PROGRAM Axes_Itp
VAR
	Fb_Axes_ItpLoadProg: ItpLoadProg;
	Fb_Axes_ItpStartStop: ItpStartStop;
	Fb_Axes_BuildItpGoup: CfgBuild3DGroup;
    localstr: STRING;
	localconstr: STRING(255);
	Fb_Axes_ItpReset_Group: ItpReset;
	
	Fb_Axes_ItpReConfig_Group: CfgReconfigGroup;
	Fb_Axes_ItpConfirmHSK: ItpConfirmHsk;
	
	M_code_rtrig: R_TRIG;
	bItpGet_MHsk: bool;
	nItp_MhskNumber: INT;
	nstep: INT;
END_VAR

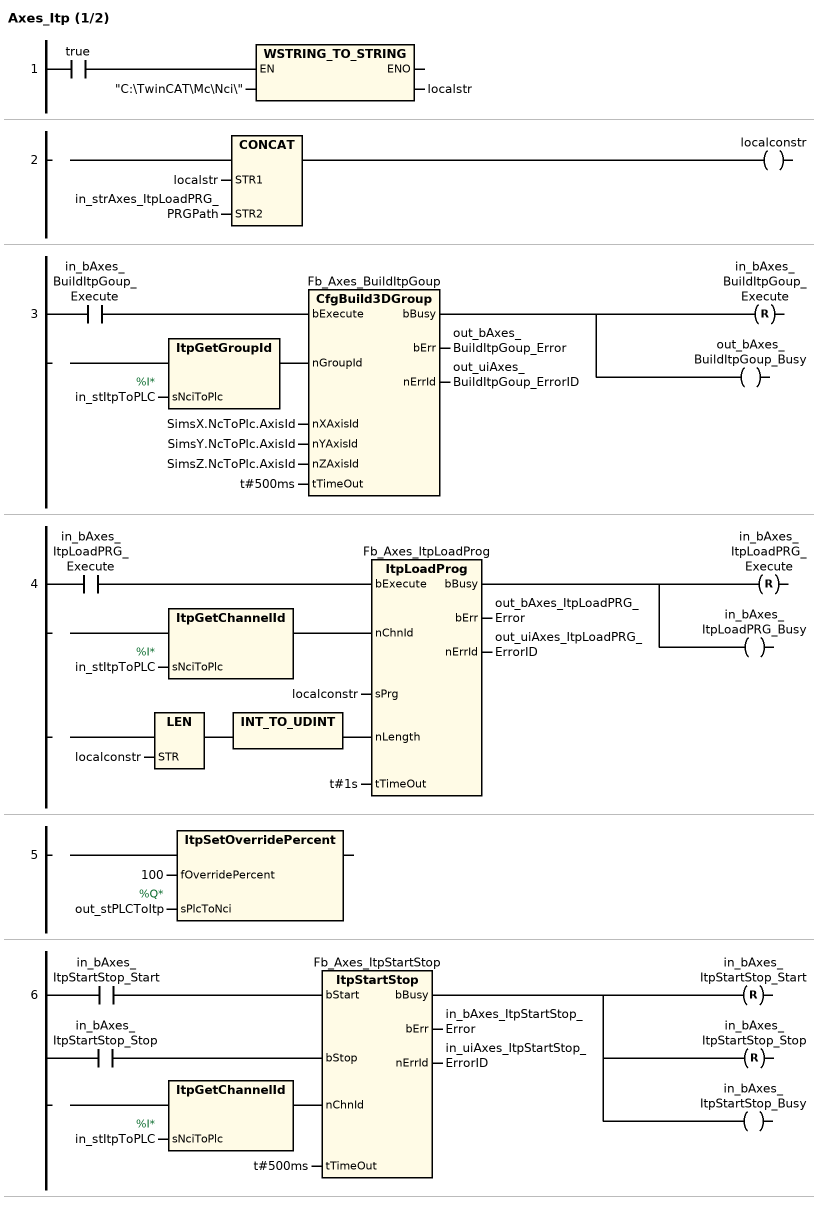
// NETWORK 1
IF true THEN localstr := WSTRING_TO_STRING("C:\TwinCAT\Mc\Nci\"); END_IF

// NETWORK 2
localconstr := CONCAT(STR1 := localstr, STR2 := in_strAxes_ItpLoadPRG_PRGPath);

// NETWORK 3
//   in_stItpToPLC: AT %I*
Fb_Axes_BuildItpGoup(
    bExecute := in_bAxes_BuildItpGoup_Execute,
    nGroupId := ItpGetGroupId(sNciToPlc := in_stItpToPLC),
    nXAxisId := SimsX.NcToPlc.AxisId,
    nYAxisId := SimsY.NcToPlc.AxisId,
    nZAxisId := SimsZ.NcToPlc.AxisId,
    tTimeOut := t#500ms,
    bErr => out_bAxes_BuildItpGoup_Error,
    nErrId => out_uiAxes_BuildItpGoup_ErrorID); // CfgBuild3DGroup
in_bAxes_BuildItpGoup_Execute R= Fb_Axes_BuildItpGoup.bBusy;
out_bAxes_BuildItpGoup_Busy := Fb_Axes_BuildItpGoup.bBusy;

// NETWORK 4
//   in_stItpToPLC: AT %I*
Fb_Axes_ItpLoadProg(
    bExecute := in_bAxes_ItpLoadPRG_Execute,
    nChnId := ItpGetChannelId(sNciToPlc := in_stItpToPLC),
    sPrg := localconstr,
    nLength := INT_TO_UDINT(LEN(STR := localconstr)),
    tTimeOut := t#1s,
    bErr => out_bAxes_ItpLoadPRG_Error,
    nErrId => out_uiAxes_ItpLoadPRG_ErrorID); // ItpLoadProg
in_bAxes_ItpLoadPRG_Execute R= Fb_Axes_ItpLoadProg.bBusy;
in_bAxes_ItpLoadPRG_Busy := Fb_Axes_ItpLoadProg.bBusy;

// NETWORK 5
//   out_stPLCToItp: AT %Q*
ItpSetOverridePercent(fOverridePercent := 100, sPlcToNci := out_stPLCToItp);

// NETWORK 6
//   in_stItpToPLC: AT %I*
Fb_Axes_ItpStartStop(
    bStart := in_bAxes_ItpStartStop_Start,
    bStop := in_bAxes_ItpStartStop_Stop,
    nChnId := ItpGetChannelId(sNciToPlc := in_stItpToPLC),
    tTimeOut := t#500ms,
    bErr => in_bAxes_ItpStartStop_Error,
    nErrId => in_uiAxes_ItpStartStop_ErrorID); // ItpStartStop
in_bAxes_ItpStartStop_Start R= Fb_Axes_ItpStartStop.bBusy;
in_bAxes_ItpStartStop_Stop R= Fb_Axes_ItpStartStop.bBusy;
in_bAxes_ItpStartStop_Busy := Fb_Axes_ItpStartStop.bBusy;

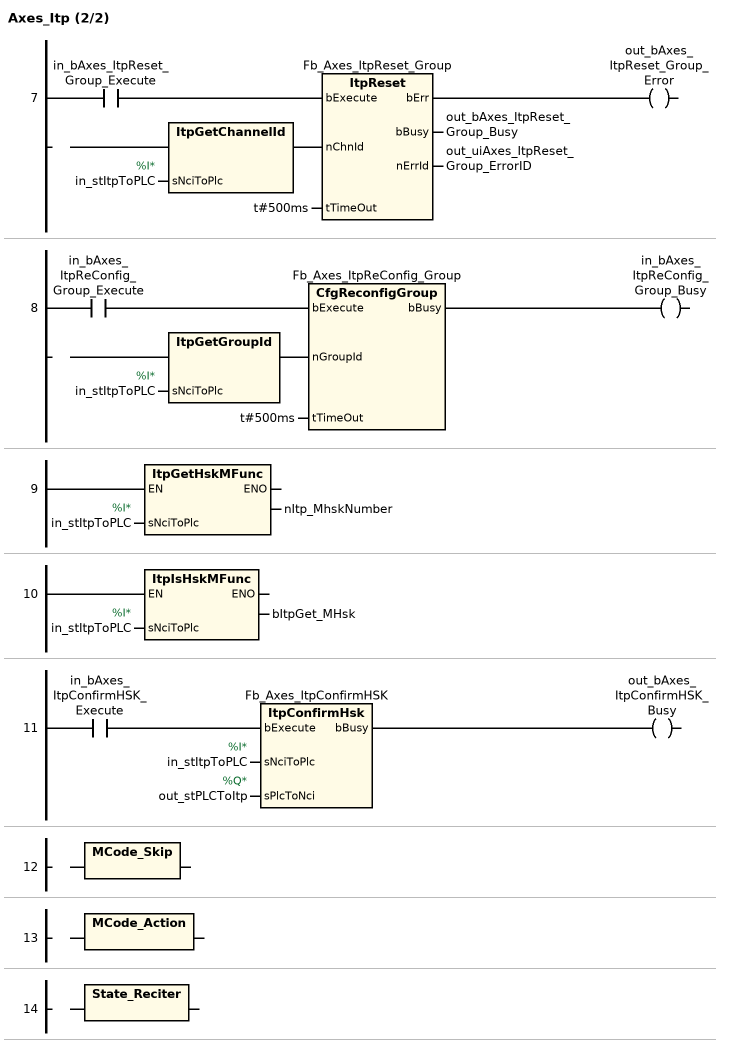
// NETWORK 7
//   in_stItpToPLC: AT %I*
Fb_Axes_ItpReset_Group(
    bExecute := in_bAxes_ItpReset_Group_Execute,
    nChnId := ItpGetChannelId(sNciToPlc := in_stItpToPLC),
    tTimeOut := t#500ms,
    bBusy => out_bAxes_ItpReset_Group_Busy,
    nErrId => out_uiAxes_ItpReset_Group_ErrorID); // ItpReset
out_bAxes_ItpReset_Group_Error := Fb_Axes_ItpReset_Group.bErr;

// NETWORK 8
//   in_stItpToPLC: AT %I*
Fb_Axes_ItpReConfig_Group(
    bExecute := in_bAxes_ItpReConfig_Group_Execute,
    nGroupId := ItpGetGroupId(sNciToPlc := in_stItpToPLC),
    tTimeOut := t#500ms); // CfgReconfigGroup
in_bAxes_ItpReConfig_Group_Busy := Fb_Axes_ItpReConfig_Group.bBusy;

// NETWORK 9
//   in_stItpToPLC: AT %I*
nItp_MhskNumber := ItpGetHskMFunc(sNciToPlc := in_stItpToPLC);

// NETWORK 10
//   in_stItpToPLC: AT %I*
bItpGet_MHsk := ItpIsHskMFunc(sNciToPlc := in_stItpToPLC);

// NETWORK 11
//   in_stItpToPLC: AT %I*
//   out_stPLCToItp: AT %Q*
Fb_Axes_ItpConfirmHSK(
    bExecute := in_bAxes_ItpConfirmHSK_Execute,
    sNciToPlc := in_stItpToPLC,
    sPlcToNci := out_stPLCToItp); // ItpConfirmHsk
out_bAxes_ItpConfirmHSK_Busy := Fb_Axes_ItpConfirmHSK.bBusy;

// NETWORK 12
MCode_Skip();

// NETWORK 13
MCode_Action();

// NETWORK 14
State_Reciter();

ACTION MCode_Action:
IF out_uiItp_Mcodenumber = 3 THEN
	out_bTOOL_HW:= TRUE;
	Axes_Itp.MCode_Skip();
END_IF

IF out_uiItp_Mcodenumber = 4 THEN
	out_bTOOL_HW:= FALSE;
	Axes_Itp.MCode_Skip();
END_IF
END_ACTION

ACTION MCode_Skip:
CASE nstep OF
	0:
		in_bAxes_ItpConfirmHSK_Execute:=FALSE;
			IF  bItpGet_MHsk AND nItp_MhskNumber =3 THEN
				nStep:=3;	
			ELSIF  bItpGet_MHsk AND nItp_MhskNumber =4 THEN
				nStep:=4;
			END_IF
	3:
		
		in_bAxes_ItpConfirmHSK_Execute:=TRUE;
			IF in_bAxes_ItpConfirmHSK_Execute AND NOT bItpGet_MHsk THEN
				nStep:=0;
			END_IF
	
	4:
		out_bTOOL_HW:= FALSE;
		in_bAxes_ItpConfirmHSK_Execute:=TRUE;
			IF in_bAxes_ItpConfirmHSK_Execute AND NOT bItpGet_MHsk THEN
				nStep:=0;
			END_IF
			
END_CASE
END_ACTION

ACTION State_Reciter:
CASE out_uiItp_InterpreterState OF
	0: out_stItp_InterpreterState_String:= "Init failed";
    1: out_stItp_InterpreterState_String:= "Idle";
    2: out_stItp_InterpreterState_String:= "Ready";
    3: out_stItp_InterpreterState_String:= "Started";
    4: out_stItp_InterpreterState_String:= "Scanning";
    5: out_stItp_InterpreterState_String:= "Running";
    6: out_stItp_InterpreterState_String:= "Stay running";
    7: out_stItp_InterpreterState_String:= "Write table";
    8: out_stItp_InterpreterState_String:= "Search line";
    9: out_stItp_InterpreterState_String:= "End";
    10:out_stItp_InterpreterState_String:= "Single Step";
    11:out_stItp_InterpreterState_String:= "Aborting";
    12:out_stItp_InterpreterState_String:= "Aborted";
    13:out_stItp_InterpreterState_String:= "Fault";
    14:out_stItp_InterpreterState_String:= "Reset";
    15:out_stItp_InterpreterState_String:= "Stop";
    16:out_stItp_InterpreterState_String:= "Wait function";
    17:out_stItp_InterpreterState_String:= "Flush buffers";
END_CASE;

IF out_wdItp_InterpolationMode=0000 THEN
	out_wdItp_InterpolationMode_string:= "Default";
    ELSIF out_wdItp_InterpolationMode=0001 THEN
    out_wdItp_InterpolationMode_string:= "SBM NC Kernel (SAF)";
    ELSIF out_wdItp_InterpolationMode=4000 THEN
    out_wdItp_InterpolationMode_string:= "SBM Block Mode Interpreter";
END_IF
END_ACTION

END_PROGRAM

(* stored: Version 1.1.0.1, ProductVersion 3.1.4018.9
   POU Axes_Itp: Id {256a6814-0e62-41a7-9557-1faae5ad7bd8}, SpecialFunc None
   Action MCode_Action: Id {561acfd1-91f0-4b52-939c-2a1dc9a4252a}
   Action MCode_Skip: Id {e92e2a65-2804-41d8-ad7b-2da571036bd8}
   Action State_Reciter: Id {2a6afd69-0c8e-4519-8e13-55d1838b361f} *)
